FUNCTION_BLOCK numeroPartidas (* Extracted Composite Function Block Type *)
  (* Standard: 61499-2 *)
  (* Version 24/02/2026 *)
  PACKAGE Hidryco.HidrycoLib;
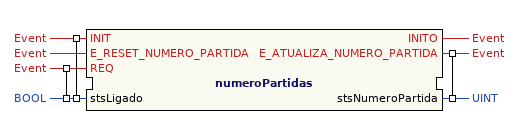
  EVENT_INPUT
    INIT WITH stsLigado; (* Service Initialization *)
    E_RESET_NUMERO_PARTIDA;
    REQ WITH stsLigado; (* Normal Execution Request *)
  END_EVENT
  EVENT_OUTPUT
    INITO; (* Initialization Confirm *)
    E_ATUALIZA_NUMERO_PARTIDA WITH stsNumeroPartida;
  END_EVENT
  VAR_INPUT
    stsLigado : BOOL;
  END_VAR
  VAR_OUTPUT
    stsNumeroPartida : UINT; (* Output event qualifier *)
  END_VAR
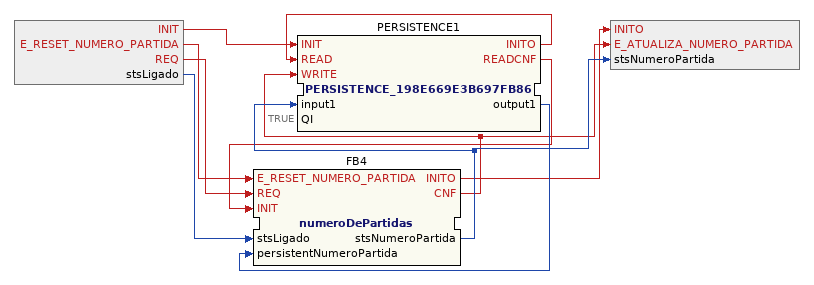
  FBS
    FB4 : numeroDePartidas;
    PERSISTENCE1 : PERSISTENCE_198E669E3B697FB86(QI := TRUE); {SET_ATTRIBUTE(Configuration.GenericFBType.InterfaceParams, Runtime.Standard#I:=1;input${I$}:UINT)}
  END_FBS
  EVENT_CONNECTIONS
    E_RESET_NUMERO_PARTIDA TO FB4.E_RESET_NUMERO_PARTIDA;
    REQ TO FB4.REQ;
    FB4.INITO TO INITO;
    FB4.CNF TO E_ATUALIZA_NUMERO_PARTIDA;
    INIT TO PERSISTENCE1.INIT;
    PERSISTENCE1.INITO TO PERSISTENCE1.READ;
    FB4.CNF TO PERSISTENCE1.WRITE;
    PERSISTENCE1.READCNF TO FB4.INIT;
  END_CONNECTIONS
  DATA_CONNECTIONS
    stsLigado TO FB4.stsLigado;
    FB4.stsNumeroPartida TO stsNumeroPartida;
    FB4.stsNumeroPartida TO PERSISTENCE1.input1;
    PERSISTENCE1.output1 TO FB4.persistentNumeroPartida;
  END_CONNECTIONS
END_FUNCTION_BLOCK
